Fanuc KAREL source: IO0118.KL

-- PROVISIONAL review KL for V1013-1; original PC SHA256 0d8f52c5e16cad9629ccf9d537ecda5c4c4397e0f9355bd3c0f6e5cdc9d1d838
-- Incomplete behavior may be omitted. Consult companion uncertainty JSON. Do not deploy.
PROGRAM IO0118
%NOLOCKGROUP
-- UNRESOLVED_LOCAL_POOL 5 cells at code offset 13; source declarations unknown
-- DIRECT_LOCAL_WORD_ACCESS alone does not prove INTEGER, REAL, or BOOLEAN
BEGIN
  -- UNRESOLVED_PC offsets 0-18; opcodes 2B,2C,7B
  -- UNRESOLVED_PC offsets 23-30; opcodes 9D,23
  -- UNRESOLVED_PC offsets 35-49; opcodes 2E,22,9D,33,35
  -- UNRESOLVED_PC offsets 54-61; opcodes 9D,23
  -- UNRESOLVED_PC offsets 66-77; opcodes 2E,23
  -- UNRESOLVED_PC offsets 82-98; opcodes 21,9D,52,19,23
  -- UNRESOLVED_PC offsets 103-107; opcodes 7F
  -- UNRESOLVED_PC offsets 112-116; opcodes 27,AA
  -- UNRESOLVED_PC offsets 121-125; opcodes 7F
END IO0118
